// TwinCAT 3 PLC project MetrisIotHub
// ProgramVersion: 3.1.4023.0
// libraries:
//   Tc2_MDP, * (Beckhoff Automation GmbH)
//   Tc2_Standard, * (Beckhoff Automation GmbH)
//   Tc2_System, * (Beckhoff Automation GmbH)
//   Tc2_Utilities, * (Beckhoff Automation GmbH)
//   Tc3_EventLogger, * (Beckhoff Automation GmbH)
//   Tc3_IotBase, * (Beckhoff Automation GmbH)
//   Tc3_JsonXml, * (Beckhoff Automation GmbH)
//   Tc3_Module, * (Beckhoff Automation GmbH)
// project tree:
//   IO/ IO.TcGVL, ST_AI_StandardChannel.TcDUT, ST_DI_StandardChannel.TcDUT, ST_AIos_Channel.TcDUT
//   / PlcTask_100ms.TcTTO, PlcTask_10ms.TcTTO, PlcTask_1ms.TcTTO
//   POUs/ Tsk_MAIN_10ms.TcPOU, Tsk_MAIN_100ms.TcPOU, Tsk_MAIN_1ms.TcPOU
// real-time tasks:
//   TASK PlcTask_10ms: cycle T#10ms, priority 8, ADS port 350
//   TASK PlcTask_1ms: cycle T#1ms, priority 4, ADS port 351
//   TASK PlcTask_100ms: cycle T#100000us, priority 10, ADS port 352
// I/O:
//   DEVICE Device 1 (EtherCAT) (disabled), AmsNetId 192.168.75.1.2.1
//     Term 1 (EK1200) [EK1200-5000 EtherCAT Power supply (2A E-Bus)]
//       Term 2 (EL3632)
//       Term 3 (EL3702) [EL3702 2Ch. Ana. Input +/-10V, DIFF, Oversample]
//       Term 4 (EL9011)
// variable links:
//   MetrisIotHub Instance <-> Device 1 (EtherCAT)/Term 1 (EK1200)/Term 2 (EL3632)
//     PlcTask_100ms Inputs/IO.AIOS[2].Raw[0] <-> Ch1 Sample 0/Ch1 Value
//   MetrisIotHub Instance <-> Device 1 (EtherCAT)/Term 1 (EK1200)/Term 3 (EL3702)
//     PlcTask_100ms Inputs/IO.AIOS[0].Raw[{0..49}] <-> Ch1 Sample {0..49}/Ch1 Value  (50 links)

CONFIGURATION MetrisIotHub
    RESOURCE PLC ON TwinCAT3
        TASK PlcTask_100ms(INTERVAL := T#100000us, PRIORITY := 10);
        TASK PlcTask_10ms(INTERVAL := T#10ms, PRIORITY := 8);
        TASK PlcTask_1ms(INTERVAL := T#1ms, PRIORITY := 4);
        PROGRAM Tsk_MAIN_100ms WITH PlcTask_100ms : Tsk_MAIN_100ms;
        PROGRAM Tsk_MAIN_10ms WITH PlcTask_10ms : Tsk_MAIN_10ms;
        PROGRAM Tsk_MAIN_1ms WITH PlcTask_1ms : Tsk_MAIN_1ms;
    END_RESOURCE
END_CONFIGURATION

// ---- IO/ST_AI_StandardChannel.TcDUT
TYPE ST_AI_StandardChannel :
STRUCT
	Status AT %I* : INT;		// channel status
	Raw AT %I*   : INT;			// raw value
	Val : REAL;					// scaled value
END_STRUCT
END_TYPE

// ---- IO/ST_DI_StandardChannel.TcDUT
TYPE ST_DI_StandardChannel :
STRUCT
	Status : INT;
	Value : INT;
END_STRUCT
END_TYPE

// ---- IO/ST_AIos_Channel.TcDUT
TYPE ST_AIos_Channel :
STRUCT
	Status AT %I*   : INT;		// channel status
	Raw AT %I*  : ARRAY[0..(IO._AIOS_NO_CHANNEL_PER_INPUT - 1)] OF INT;			// raw value
	Val : ARRAY[0..(IO._AIOS_NO_CHANNEL_PER_INPUT - 1)] OF REAL;				// scaled value
END_STRUCT
END_TYPE

// ---- IO/IO.TcGVL
{attribute 'global_init_slot' := '40500'}

// INPUT DESIGNATION:
// - DI - digital input
//		- mapping to MAIN task

// - AI - analog input
//		- mapping to MAIN task 

// - AIOS - analog input with oversampling
//		- mapping to MAIN_HS task with 1ms cycle time 
//		- recorded into FiFo buffer to be handled by slow task

VAR_GLOBAL CONSTANT
	// Standard AI configuration
	_AI_NO_INPUTS : UDINT := 10;						// number of physical input	

	// Standard DI configuration
	_DI_NO_INPUTS : UDINT := 10;						// number of physical input	

	// Standard DQ configuration
	_DQ_NO_INPUTS : UDINT := 10;						// number of physical output	

	
	_AIOS_NO_INPUTS	: UDINT := 3;						// number of physical input 
	_AIOS_NO_CHANNEL_PER_INPUT : UDINT := 50;			// Number of channels for single input, oversampling factor 10 - 50
	
	// Max number of samples
	_AIOS_SAMPLE_RATE : UDINT := _AIOS_NO_CHANNEL_PER_INPUT * 1000;			// Number of sampoles per sec := Oversampling * HS cycle per sec
	
END_VAR


{attribute 'qualified_only'}
VAR_GLOBAL

	AIOS : ARRAY[0..(_AIOS_NO_INPUTS)] OF  ST_AIOS_Channel;
	
	AI : ARRAY[0..(_AI_NO_INPUTS)] OF ST_AI_StandardChannel;
	
	DI AT %I* : ARRAY[0..(_DI_NO_INPUTS)] OF ST_DI_StandardChannel;

	DQ AT %Q* : ARRAY[0..(_DQ_NO_INPUTS)] OF BOOL;

	
END_VAR

// ---- POUs/Tsk_MAIN_100ms.TcPOU
PROGRAM Tsk_MAIN_100ms
VAR

END_VAR

END_PROGRAM

// ---- POUs/Tsk_MAIN_10ms.TcPOU
PROGRAM Tsk_MAIN_10ms
VAR

END_VAR

END_PROGRAM

// ---- POUs/Tsk_MAIN_1ms.TcPOU
PROGRAM Tsk_MAIN_1ms
VAR


END_VAR

END_PROGRAM
